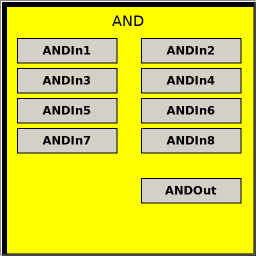
VISUALIZATION V_PH_AND  // 256x256
VAR_INPUT
	stSafetyAnd			:ST_SAFETY_FBAND;
END_VAR
    Rectangle (2,2 256x256), colour toggle: stSafetyAnd.bGeneralError
    RoundedRectangle (17,68 100x25), "ANDIn3", colour toggle: stSafetyAnd.uStatus.stStatusWords.wInputs.1
    RoundedRectangle (141,68 100x25), "ANDIn4", colour toggle: stSafetyAnd.uStatus.stStatusWords.wInputs.11
    RoundedRectangle (141,98 100x25), "ANDIn6", colour toggle: stSafetyAnd.uStatus.stStatusWords.wInputs.13
    RoundedRectangle (141,38 100x25), "ANDIn2", colour toggle: stSafetyAnd.uStatus.stStatusWords.wInputs.9
    RoundedRectangle (17,98 100x25), "ANDIn5", colour toggle: stSafetyAnd.uStatus.stStatusWords.wInputs.12
    RoundedRectangle (141,128 100x25), "ANDIn8", colour toggle: stSafetyAnd.uStatus.stStatusWords.wInputs.15
    RoundedRectangle (17,128 100x25), "ANDIn7", colour toggle: stSafetyAnd.uStatus.stStatusWords.wInputs.14
    RoundedRectangle (141,178 100x25), "ANDOut", colour toggle: stSafetyAnd.uStatus.stStatusWords.wOutputs.0
    RoundedRectangle (17,38 100x25), "ANDIn1", colour toggle: stSafetyAnd.uStatus.stStatusWords.wInputs.8
    Label (53,6 150x30), "AND"
    Textfield (17,226 234x25), text list: 'TL_FbState', text index: stSafetyAnd.eState
END_VISUALIZATION

(* stored: Version 1.1.0.1, ProductVersion 3.1.4024.4
   Visu V_PH_AND: Id {5570644b-80d3-4fc9-af7f-6d54ca56f261} *)
